// TIA Portal V18 export
FUNCTION_BLOCK "Utility_selection"   // FB7, FBD
TITLE = Selection1_12 , flushing13
{ S7_Optimized_Access := 'TRUE' }
VERSION : 0.1
// stored: AutoNumber false, IsIECCheckEnabled false, IsRetainMemResEnabled false, MemoryReserve 100, SetENOAutomatically false, UDAEnableTagReadback false
   VAR_INPUT
      utl_type : Int;
      chbs_ofb : Bool;
      chbs_cfb : Bool;
      chws_ofb : Bool;
      chws_cfb : Bool;
      cws_ofb : Bool;
      cws_cfb : Bool;
      hws_ofb : Bool;
      hws_cfb : Bool;
      as_ofb : Bool;
      as_cfb : Bool;
      byp_ofb : Bool;
      byp_cfb : Bool;
      chbr_ofb : Bool;
      chbr_cfb : Bool;
      chwr_ofb : Bool;
      chwr_cfb : Bool;
      hwr_ofb : Bool;
      hwr_cfb : Bool;
      cwr_ofb : Bool;
      cwr_cfb : Bool;
      cond_ofb : Bool;
      cond_cfb : Bool;
      dr_ofb : Bool;
      dr_cfb : Bool;
      av_ofb : Bool;
      av_cfb : Bool;
      scv_ofb : Bool;
      times : Array[0..2] of DInt;
   END_VAR
   VAR_OUTPUT
      chbs_cmd : Bool;
      chws_cmd : Bool;
      cws_cmd : Bool;
      hws_cmd : Bool;
      as_cmd : Bool;
      byp_cmd : Bool;
      chbr_cmd : Bool;
      chwr_cmd : Bool;
      cwr_cmd : Bool;
      hwr_cmd : Bool;
      cond_cmd : Bool;
      dr_cmd : Bool;
      av_cmd : Bool;
      scv_cmd : Bool;
      flush_time : DInt;
      vent_time : DInt;
      drine_time : DInt;
      CMNR_cmd : Bool;
   END_VAR
   VAR_IN_OUT
      control { ExternalVisible := 'False'} : Word;
      utl_bit : Bool;
   END_VAR
   VAR
      selection : Int;
      br_sel : Bool;
      chw_sel : Bool;
      cw_sel : Bool;
      hw_sel : Bool;
      flush_sel : Bool;
      st_sel : Bool;
      prev_util : Int;
      vent_start : Bool;
      start_temp : Bool;
      start : Bool;
      flush_tm_comp : Bool;
      am : Bool;
      pause : Bool;
      chbr_cmd1 : Bool;
      chbr_cmd2 : Bool;
      agr_fail : Bool;
      hold : Bool;
      hold_t : Bool;
      status : Word;
      steam_flush : Bool;
      SUV_flush : Bool;
      Pres_low : Bool;
      uti_cv : Bool;
      hw_autoflush : Bool;
      emstop : Bool;
      temp : Bool;
      en_flush : Bool;
      dr_start : Bool;
      hwr_cmd1 : Bool;
      hwr_cmd2 : Bool;
      chwr_cmd1 : Bool;
      chwr_cmd2 : Bool;
      cond_cmd1 : Bool;
      cwr_cmd1 : Bool;
      cwr_cmd2 : Bool;
      br_flush : Bool;
      chw_flush : Bool;
      cw_flush : Bool;
      hw_flush : Bool;
      st_flush : Bool;
      byp_cmd2 : Bool;
      Flush_Dint : DInt;
      Flush_Ptime : Time;
      Flush_Etime : Time;
      Flush_TTime : DInt;
      Vent_Etime : Time;
      Vent_TTime : DInt;
      Vent_Ptime : Time;
      Vent_Dint : DInt;
      Cond_Dint : DInt;
      Cond_Ptime : Time;
      Cond_Etime : Time;
      Cond_TTime : DInt;
      reserved : Bool;
      Vent_tm_comp : Bool;
      Cond_tm_comp : Bool;
      US_TOF3 { S7_SetPoint := 'True'} : TOF_TIME;
      US_TON2 { S7_SetPoint := 'True'} : TON_TIME;
      US_TON3 { S7_SetPoint := 'True'} : TON_TIME;
      US_TON4 { S7_SetPoint := 'True'} : TON_TIME;
      US_TON5 { S7_SetPoint := 'True'} : TON_TIME;
      US_TP2 { S7_SetPoint := 'True'} : TP_TIME;
      US_TP3 { S7_SetPoint := 'True'} : TP_TIME;
      US_TP4 { S7_SetPoint := 'True'} : TP_TIME;
      US_TOF1 { S7_SetPoint := 'True'} : TOF_TIME;
      UP_TP6 { S7_SetPoint := 'True'} : TP_TIME;
      US_TP8 { S7_SetPoint := 'True'} : TP_TIME;
      US_TP7 { S7_SetPoint := 'True'} : TP_TIME;
      US_TP9 { S7_SetPoint := 'True'} : TP_TIME;
      UP_TP1 { S7_SetPoint := 'True'} : TP_TIME;
      US_TP10 { S7_SetPoint := 'True'} : TP_TIME;
      US_TOF2 { S7_SetPoint := 'True'} : TOF_TIME;
      US_TOF4 { S7_SetPoint := 'True'} : TOF_TIME;
      US_TOF6 { S7_SetPoint := 'True'} : TOF_TIME;
      US_TP11 { S7_SetPoint := 'True'} : TP_TIME;
      US_TP12 { S7_SetPoint := 'True'} : TP_TIME;
      US_TON6 { S7_SetPoint := 'True'} : TON_TIME;
      US_TP5 { S7_SetPoint := 'True'} : TP_TIME;
      US_TON7 { S7_SetPoint := 'True'} : TON_TIME;
      US_TP13 { S7_SetPoint := 'True'} : TP_TIME;
      US_TP14 { S7_SetPoint := 'True'} : TP_TIME;
      US_TON8 { S7_SetPoint := 'True'} : TON_TIME;
      US_TP15 { S7_SetPoint := 'True'} : TP_TIME;
      US_TP20 { S7_SetPoint := 'True'} : TP_TIME;
      US_TON10 { S7_SetPoint := 'True'} : TON_TIME;
      US_TP16 { S7_SetPoint := 'True'} : TP_TIME;
      US_TON9 { S7_SetPoint := 'True'} : TON_TIME;
      US_TP17 { S7_SetPoint := 'True'} : TP_TIME;
      US_TP21 { S7_SetPoint := 'True'} : TP_TIME;
      S_TON11 { S7_SetPoint := 'True'} : TON_TIME;
      US_TP18 { S7_SetPoint := 'True'} : TP_TIME;
      US_TP19 { S7_SetPoint := 'True'} : TP_TIME;
   END_VAR
   VAR_TEMP   // added for the SCL form of the ladder/FBD networks
      _w1 : Bool;
   END_VAR
BEGIN

REGION Network 1: utility selection and moving
   // utility selection and moving
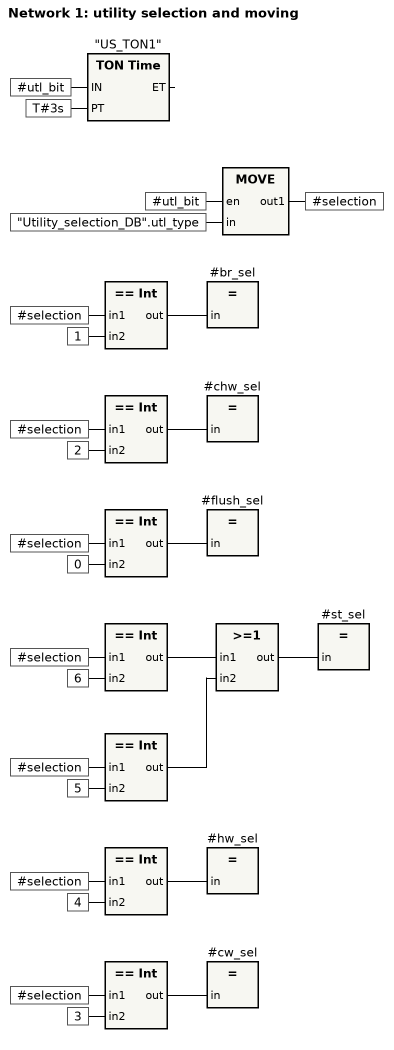
   "US_TON1".TON(IN := #utl_bit, PT := T#3s);
   IF #utl_bit THEN #selection := "Utility_selection_DB".utl_type; END_IF;
   #br_sel := #selection = 1;
   #chw_sel := #selection = 2;
   #flush_sel := #selection = 0;
   #st_sel := (#selection = 6) OR (#selection = 5);
   #hw_sel := #selection = 4;
   #cw_sel := #selection = 3;
END_REGION

REGION Network 2: previous utiliy identifucation
   // previous utiliy identifucation
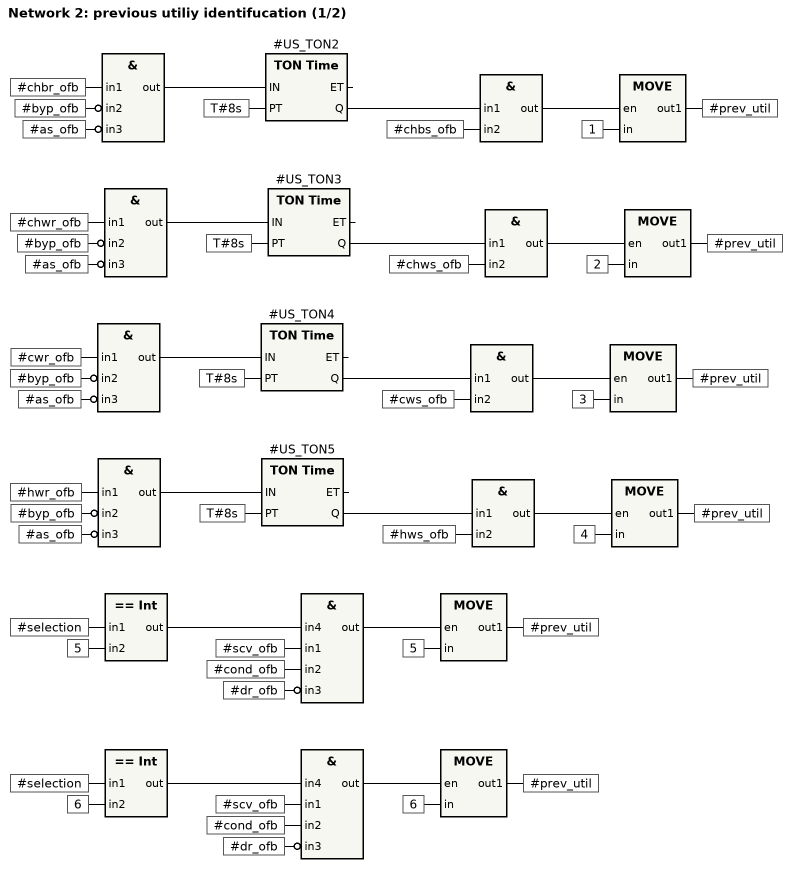
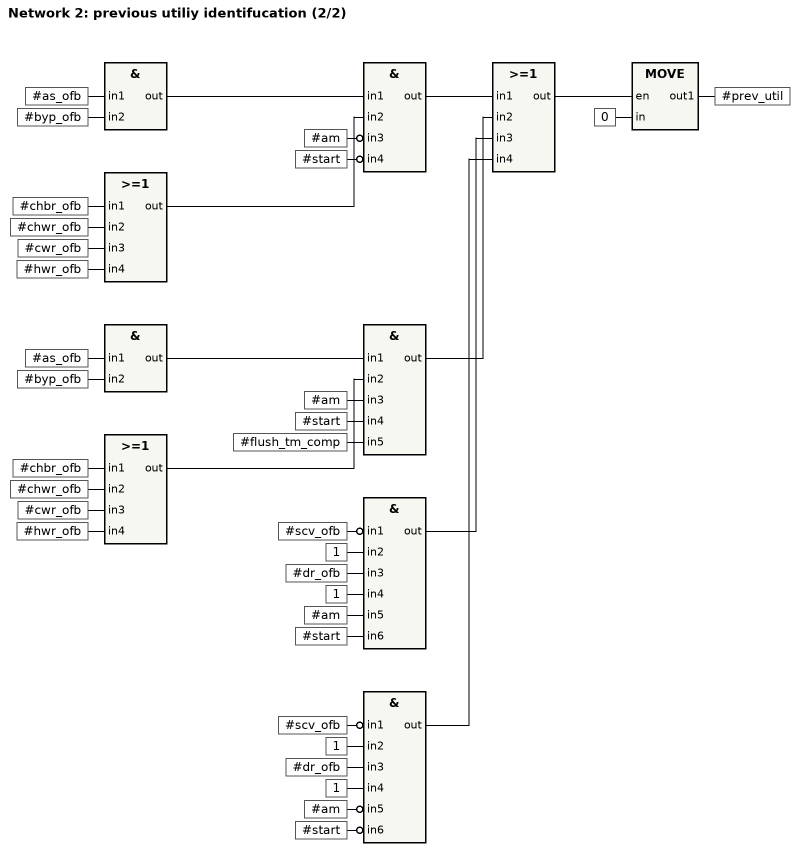
   #US_TON2(IN := #chbr_ofb AND NOT #byp_ofb AND NOT #as_ofb, PT := T#8s);   // TON
   IF #US_TON2.Q AND #chbs_ofb THEN #prev_util := 1; END_IF;
   #US_TON3(IN := #chwr_ofb AND NOT #byp_ofb AND NOT #as_ofb, PT := T#8s);   // TON
   IF #US_TON3.Q AND #chws_ofb THEN #prev_util := 2; END_IF;
   #US_TON4(IN := #cwr_ofb AND NOT #byp_ofb AND NOT #as_ofb, PT := T#8s);   // TON
   IF #US_TON4.Q AND #cws_ofb THEN #prev_util := 3; END_IF;
   #US_TON5(IN := #hwr_ofb AND NOT #byp_ofb AND NOT #as_ofb, PT := T#8s);   // TON
   IF #US_TON5.Q AND #hws_ofb THEN #prev_util := 4; END_IF;
   IF (#selection = 5) AND #scv_ofb AND #cond_ofb AND NOT #dr_ofb THEN #prev_util := 5; END_IF;
   IF (#selection = 6) AND #scv_ofb AND #cond_ofb AND NOT #dr_ofb THEN #prev_util := 6; END_IF;
   IF (#as_ofb AND #byp_ofb AND (#chbr_ofb OR #chwr_ofb OR #cwr_ofb OR #hwr_ofb) AND NOT #am AND NOT #start) OR (#as_ofb AND #byp_ofb AND (#chbr_ofb OR #chwr_ofb OR #cwr_ofb OR #hwr_ofb) AND #am AND #start AND #flush_tm_comp) OR (NOT #scv_ofb AND 1 AND #dr_ofb AND 1 AND #am AND #start) OR (NOT #scv_ofb AND 1 AND #dr_ofb AND 1 AND NOT #am AND NOT #start) THEN
       #prev_util := 0;
   END_IF;
END_REGION

REGION Network 3: flushing Identification
   // flushing Identification
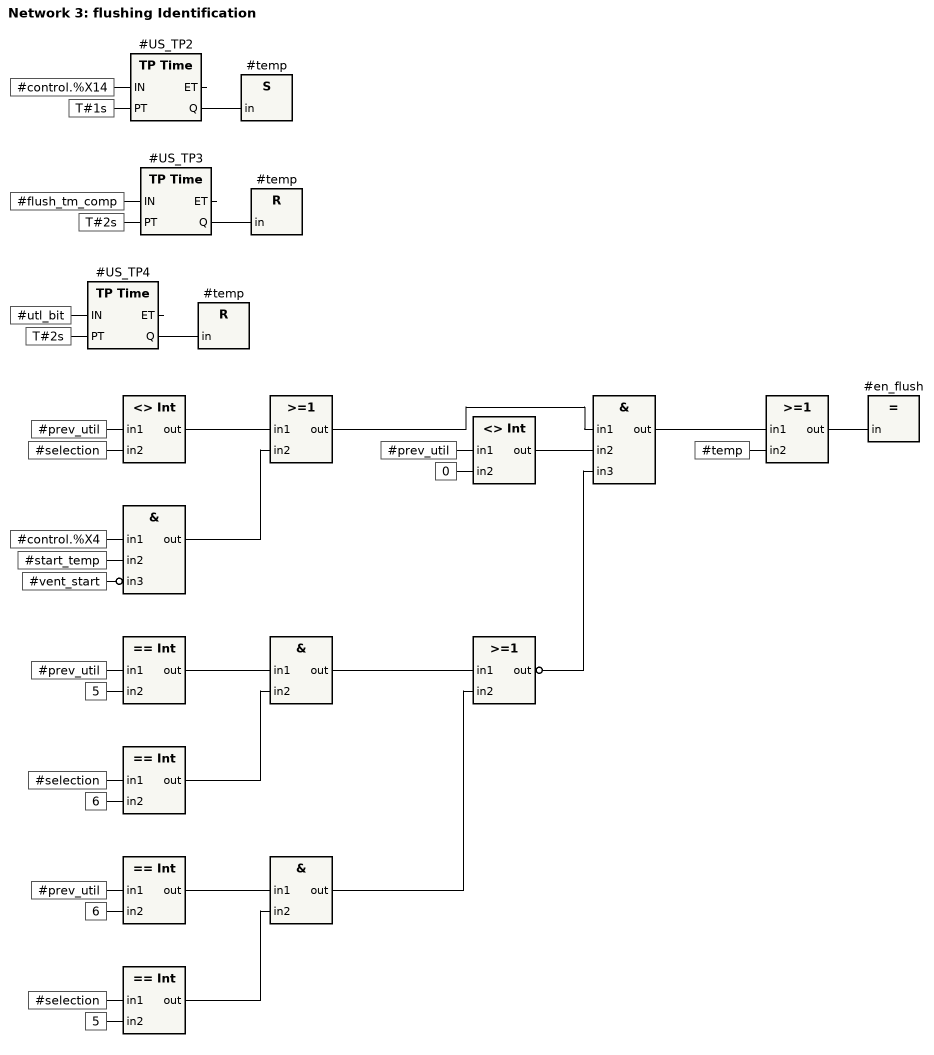
   #US_TP2(IN := #control.%X14, PT := T#1s);   // TP
   IF #US_TP2.Q THEN #temp := TRUE; END_IF;
   #US_TP3(IN := #flush_tm_comp, PT := T#2s);   // TP
   IF #US_TP3.Q THEN #temp := FALSE; END_IF;
   #US_TP4(IN := #utl_bit, PT := T#2s);   // TP
   IF #US_TP4.Q THEN #temp := FALSE; END_IF;
   #en_flush := (((#prev_util <> #selection) OR (#control.%X4 AND #start_temp AND NOT #vent_start)) AND (#prev_util <> 0) AND NOT (((#prev_util = 5) AND (#selection = 6)) OR ((#prev_util = 6) AND (#selection = 5)))) OR #temp;
END_REGION

REGION Network 4: temp_start
   // temp_start
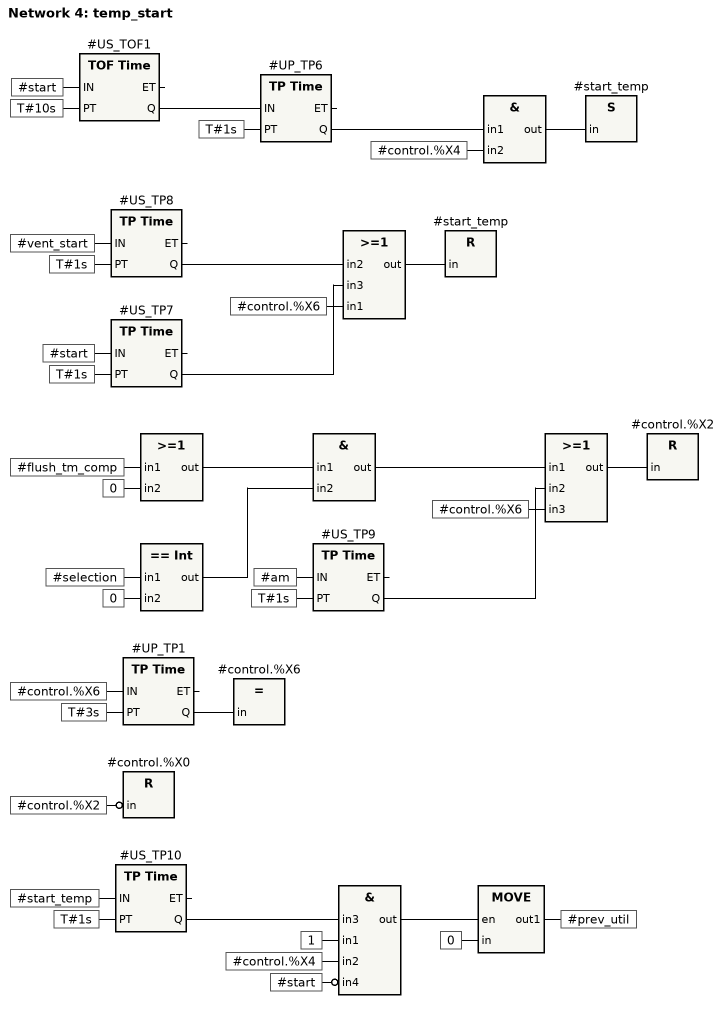
   #US_TOF1(IN := #start, PT := T#10s);   // TOF
   #UP_TP6(IN := #US_TOF1.Q, PT := T#1s);   // TP
   IF #UP_TP6.Q AND #control.%X4 THEN #start_temp := TRUE; END_IF;
   #US_TP8(IN := #vent_start, PT := T#1s);   // TP
   #US_TP7(IN := #start, PT := T#1s);   // TP
   IF #US_TP8.Q OR #US_TP7.Q OR #control.%X6 THEN #start_temp := FALSE; END_IF;
   #US_TP9(IN := #am, PT := T#1s);   // TP
   IF ((#flush_tm_comp OR 0) AND (#selection = 0)) OR #US_TP9.Q OR #control.%X6 THEN
       #control.%X2 := FALSE;
   END_IF;
   #UP_TP1(IN := #control.%X6, PT := T#3s);   // TP
   #control.%X6 := #UP_TP1.Q;
   IF NOT #control.%X2 THEN #control.%X0 := FALSE; END_IF;
   #US_TP10(IN := #start_temp, PT := T#1s);   // TP
   IF #US_TP10.Q AND 1 AND #control.%X4 AND NOT #start THEN #prev_util := 0; END_IF;
END_REGION

REGION Network 5: control and status word
   // control and status word
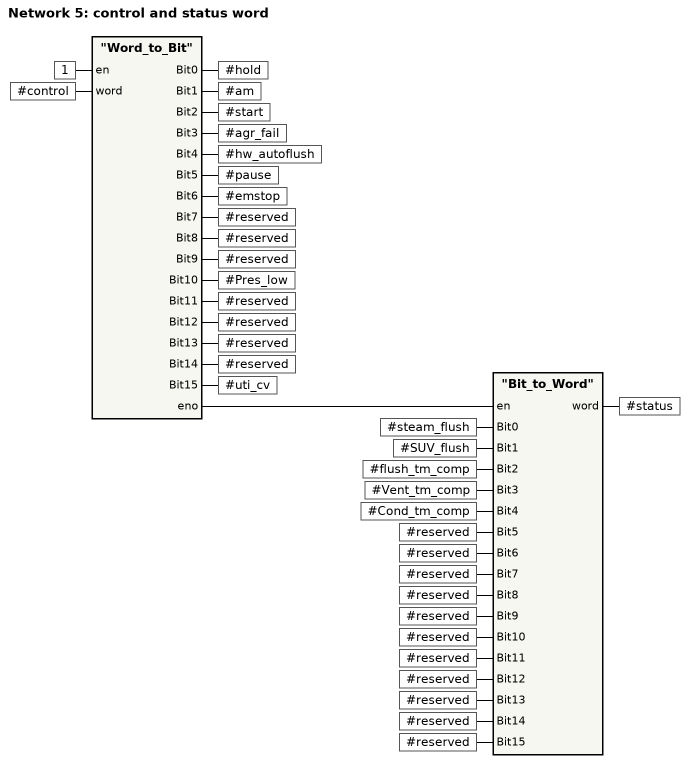
   "Word_to_Bit"(EN := 1,
                 "word" := #control,
                 Bit0 => #hold,
                 Bit1 => #am,
                 Bit2 => #start,
                 Bit3 => #agr_fail,
                 Bit4 => #hw_autoflush,
                 Bit5 => #pause,
                 Bit6 => #emstop,
                 Bit7 => #reserved,
                 Bit8 => #reserved,
                 Bit9 => #reserved,
                 Bit10 => #Pres_low,
                 Bit11 => #reserved,
                 Bit12 => #reserved,
                 Bit13 => #reserved,
                 Bit14 => #reserved,
                 Bit15 => #uti_cv,
                 ENO => #_w1);
   IF #_w1 THEN
       "Bit_to_Word"(Bit0 := #steam_flush,
                     Bit1 := #SUV_flush,
                     Bit2 := #flush_tm_comp,
                     Bit3 := #Vent_tm_comp,
                     Bit4 := #Cond_tm_comp,
                     Bit5 := #reserved,
                     Bit6 := #reserved,
                     Bit7 := #reserved,
                     Bit8 := #reserved,
                     Bit9 := #reserved,
                     Bit10 := #reserved,
                     Bit11 := #reserved,
                     Bit12 := #reserved,
                     Bit13 := #reserved,
                     Bit14 := #reserved,
                     Bit15 := #reserved,
                     "word" => #status);
   END_IF;
END_REGION

REGION Network 6: Brine select
   // Brine select
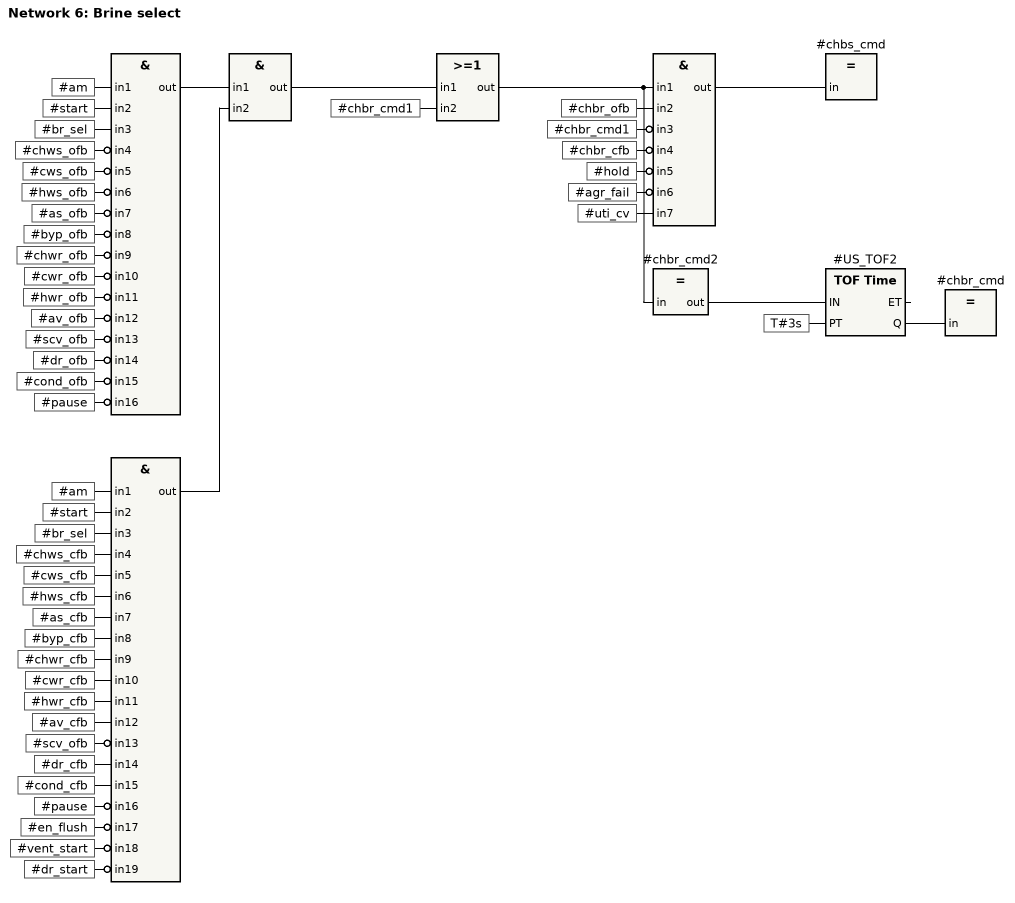
   #_w1 := (#am AND #start AND #br_sel AND NOT #chws_ofb AND NOT #cws_ofb AND NOT #hws_ofb AND NOT #as_ofb AND NOT #byp_ofb AND NOT #chwr_ofb AND NOT #cwr_ofb AND NOT #hwr_ofb AND NOT #av_ofb AND NOT #scv_ofb AND NOT #dr_ofb AND NOT #cond_ofb AND NOT #pause AND #am AND #start AND #br_sel AND #chws_cfb AND #cws_cfb AND #hws_cfb AND #as_cfb AND #byp_cfb AND #chwr_cfb AND #cwr_cfb AND #hwr_cfb AND #av_cfb AND NOT #scv_ofb AND #dr_cfb AND #cond_cfb AND NOT #pause AND NOT #en_flush AND NOT #vent_start AND NOT #dr_start) OR #chbr_cmd1;
   #chbs_cmd := #_w1 AND #chbr_ofb AND NOT #chbr_cmd1 AND NOT #chbr_cfb AND NOT #hold AND NOT #agr_fail AND #uti_cv;
   #chbr_cmd2 := #_w1;
   #US_TOF2(IN := #_w1, PT := T#3s);   // TOF
   #chbr_cmd := #US_TOF2.Q;
END_REGION

REGION Network 7: CMNR logic
   // CMNR logic
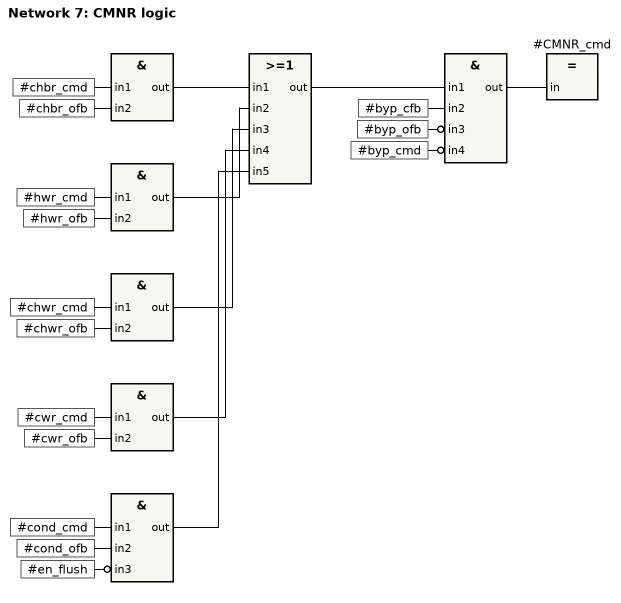
   #CMNR_cmd := ((#chbr_cmd AND #chbr_ofb) OR (#hwr_cmd AND #hwr_ofb) OR (#chwr_cmd AND #chwr_ofb) OR (#cwr_cmd AND #cwr_ofb) OR (#cond_cmd AND #cond_ofb AND NOT #en_flush)) AND #byp_cfb AND NOT #byp_ofb AND NOT #byp_cmd;
END_REGION

REGION Network 8: HW select
   // Hw select
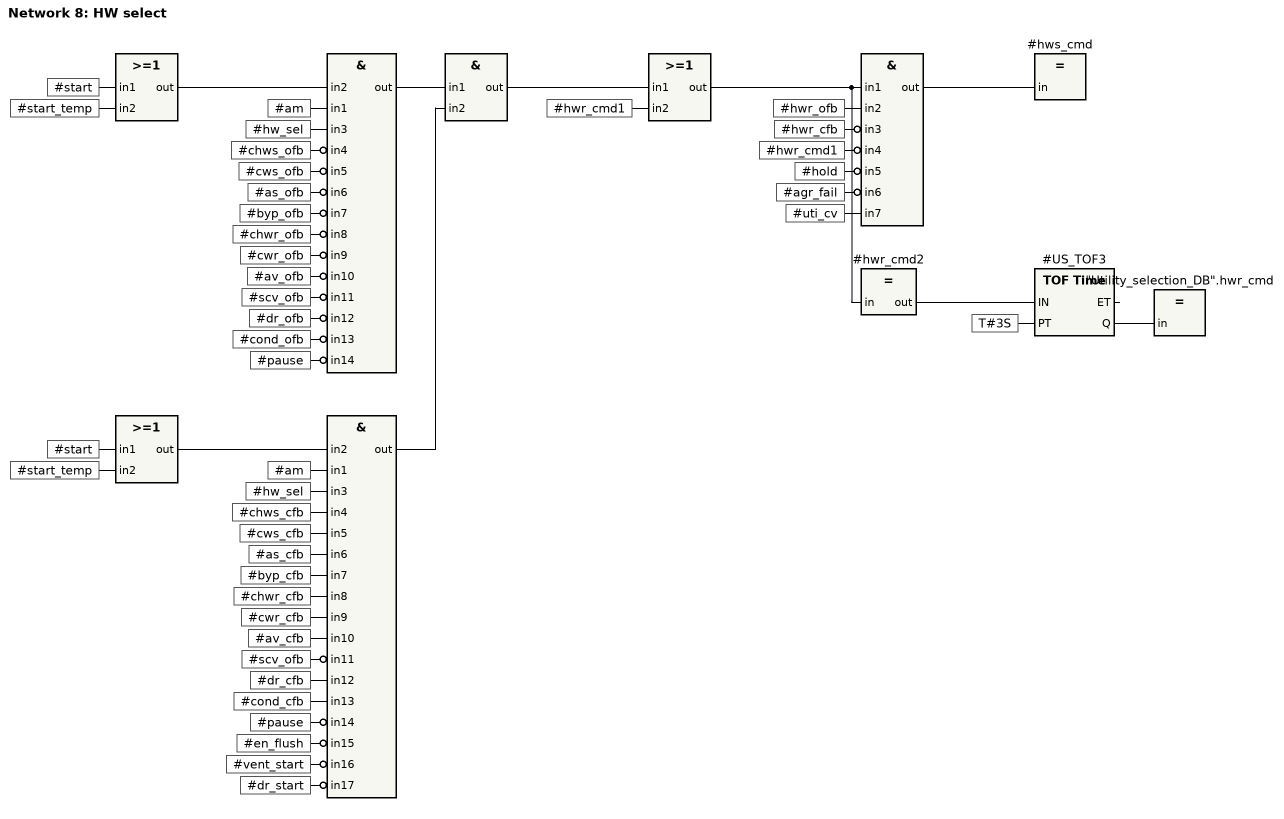
   #_w1 := ((#start OR #start_temp) AND #am AND #hw_sel AND NOT #chws_ofb AND NOT #cws_ofb AND NOT #as_ofb AND NOT #byp_ofb AND NOT #chwr_ofb AND NOT #cwr_ofb AND NOT #av_ofb AND NOT #scv_ofb AND NOT #dr_ofb AND NOT #cond_ofb AND NOT #pause AND (#start OR #start_temp) AND #am AND #hw_sel AND #chws_cfb AND #cws_cfb AND #as_cfb AND #byp_cfb AND #chwr_cfb AND #cwr_cfb AND #av_cfb AND NOT #scv_ofb AND #dr_cfb AND #cond_cfb AND NOT #pause AND NOT #en_flush AND NOT #vent_start AND NOT #dr_start) OR #hwr_cmd1;
   #hws_cmd := #_w1 AND #hwr_ofb AND NOT #hwr_cfb AND NOT #hwr_cmd1 AND NOT #hold AND NOT #agr_fail AND #uti_cv;
   #hwr_cmd2 := #_w1;
   #US_TOF3(IN := #_w1, PT := T#3S);   // TOF
   "Utility_selection_DB".hwr_cmd := #US_TOF3.Q;
END_REGION

REGION Network 9: chw select
   // chw select
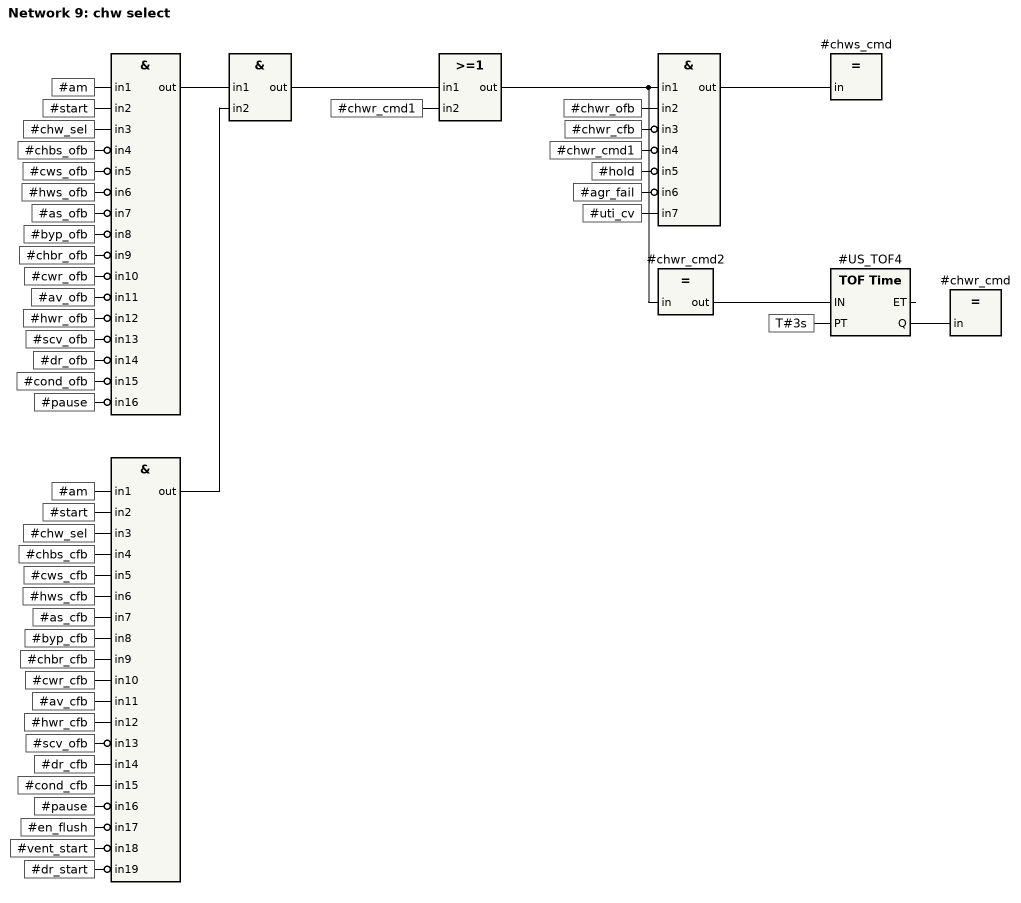
   #_w1 := (#am AND #start AND #chw_sel AND NOT #chbs_ofb AND NOT #cws_ofb AND NOT #hws_ofb AND NOT #as_ofb AND NOT #byp_ofb AND NOT #chbr_ofb AND NOT #cwr_ofb AND NOT #av_ofb AND NOT #hwr_ofb AND NOT #scv_ofb AND NOT #dr_ofb AND NOT #cond_ofb AND NOT #pause AND #am AND #start AND #chw_sel AND #chbs_cfb AND #cws_cfb AND #hws_cfb AND #as_cfb AND #byp_cfb AND #chbr_cfb AND #cwr_cfb AND #av_cfb AND #hwr_cfb AND NOT #scv_ofb AND #dr_cfb AND #cond_cfb AND NOT #pause AND NOT #en_flush AND NOT #vent_start AND NOT #dr_start) OR #chwr_cmd1;
   #chws_cmd := #_w1 AND #chwr_ofb AND NOT #chwr_cfb AND NOT #chwr_cmd1 AND NOT #hold AND NOT #agr_fail AND #uti_cv;
   #chwr_cmd2 := #_w1;
   #US_TOF4(IN := #_w1, PT := T#3s);   // TOF
   #chwr_cmd := #US_TOF4.Q;
END_REGION

REGION Network 10: Steam select
   // Steam select
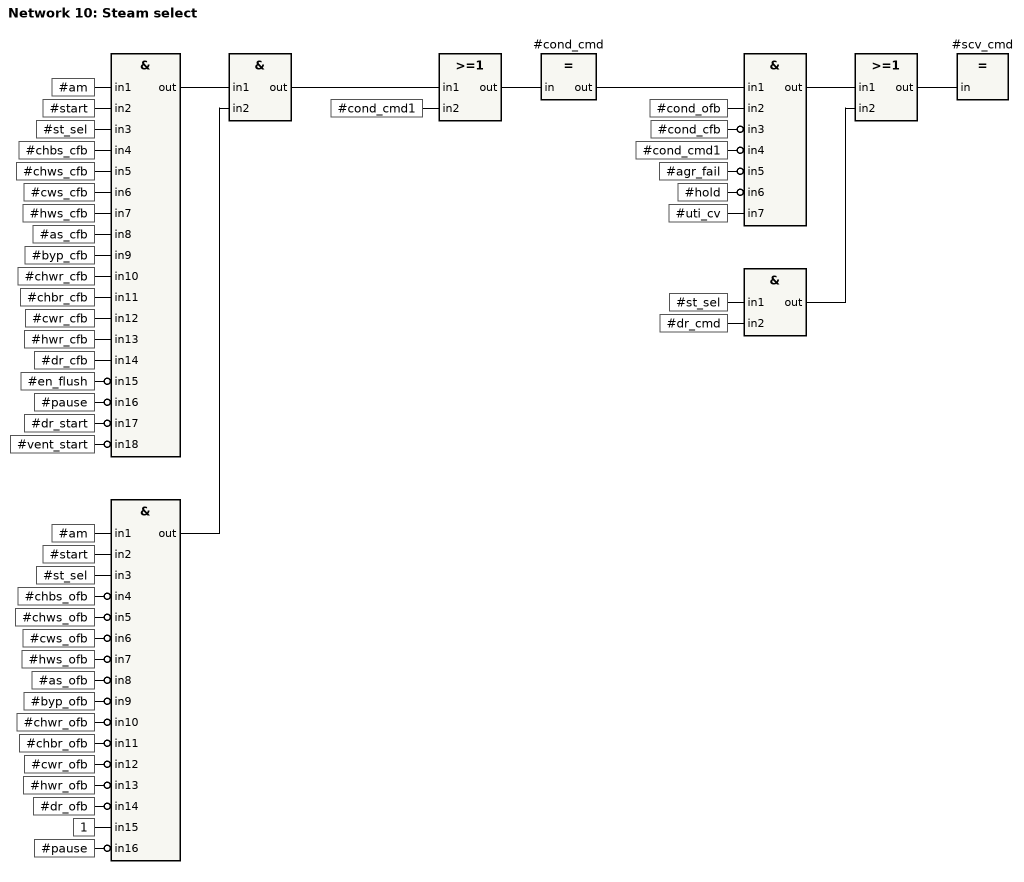
   #cond_cmd := (#am AND #start AND #st_sel AND #chbs_cfb AND #chws_cfb AND #cws_cfb AND #hws_cfb AND #as_cfb AND #byp_cfb AND #chwr_cfb AND #chbr_cfb AND #cwr_cfb AND #hwr_cfb AND #dr_cfb AND NOT #en_flush AND NOT #pause AND NOT #dr_start AND NOT #vent_start AND #am AND #start AND #st_sel AND NOT #chbs_ofb AND NOT #chws_ofb AND NOT #cws_ofb AND NOT #hws_ofb AND NOT #as_ofb AND NOT #byp_ofb AND NOT #chwr_ofb AND NOT #chbr_ofb AND NOT #cwr_ofb AND NOT #hwr_ofb AND NOT #dr_ofb AND 1 AND NOT #pause) OR #cond_cmd1;
   #scv_cmd := (#cond_cmd AND #cond_ofb AND NOT #cond_cfb AND NOT #cond_cmd1 AND NOT #agr_fail AND NOT #hold AND #uti_cv) OR (#st_sel AND #dr_cmd);
END_REGION

REGION Network 11: cw_select
   // cw_select
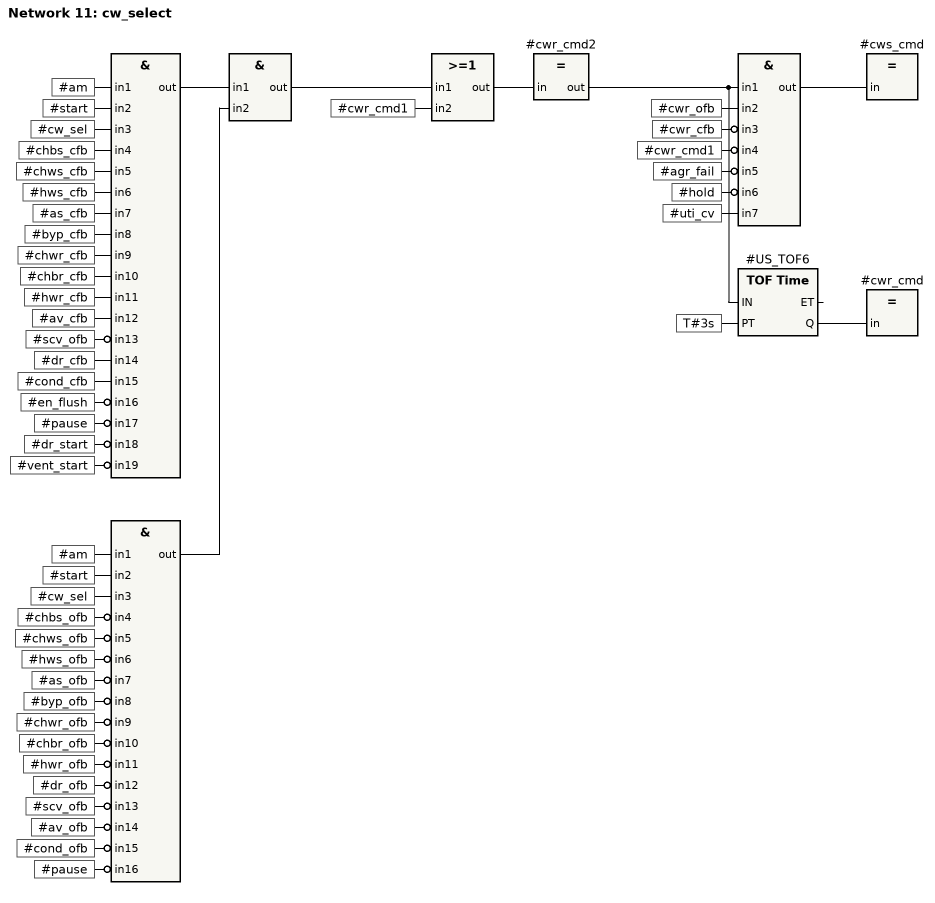
   #cwr_cmd2 := (#am AND #start AND #cw_sel AND #chbs_cfb AND #chws_cfb AND #hws_cfb AND #as_cfb AND #byp_cfb AND #chwr_cfb AND #chbr_cfb AND #hwr_cfb AND #av_cfb AND NOT #scv_ofb AND #dr_cfb AND #cond_cfb AND NOT #en_flush AND NOT #pause AND NOT #dr_start AND NOT #vent_start AND #am AND #start AND #cw_sel AND NOT #chbs_ofb AND NOT #chws_ofb AND NOT #hws_ofb AND NOT #as_ofb AND NOT #byp_ofb AND NOT #chwr_ofb AND NOT #chbr_ofb AND NOT #hwr_ofb AND NOT #dr_ofb AND NOT #scv_ofb AND NOT #av_ofb AND NOT #cond_ofb AND NOT #pause) OR #cwr_cmd1;
   #cws_cmd := #cwr_cmd2 AND #cwr_ofb AND NOT #cwr_cfb AND NOT #cwr_cmd1 AND NOT #agr_fail AND NOT #hold AND #uti_cv;
   #US_TOF6(IN := #cwr_cmd2, PT := T#3s);   // TOF
   #cwr_cmd := #US_TOF6.Q;
END_REGION

REGION Network 12: flush selection
   // flush selection
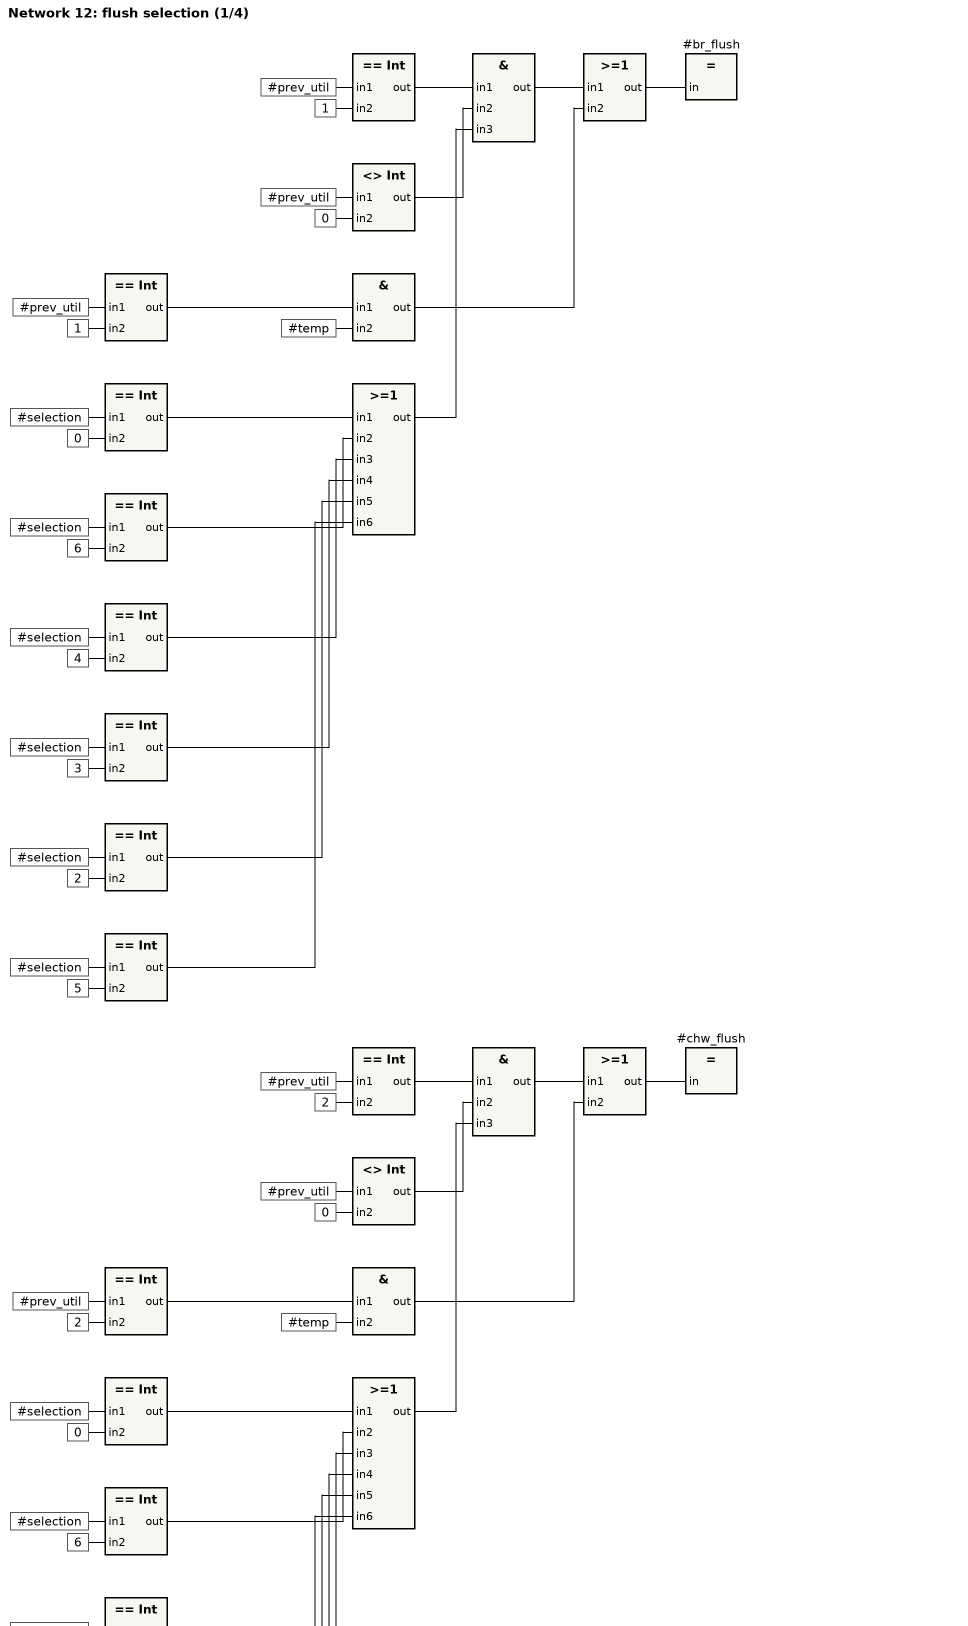
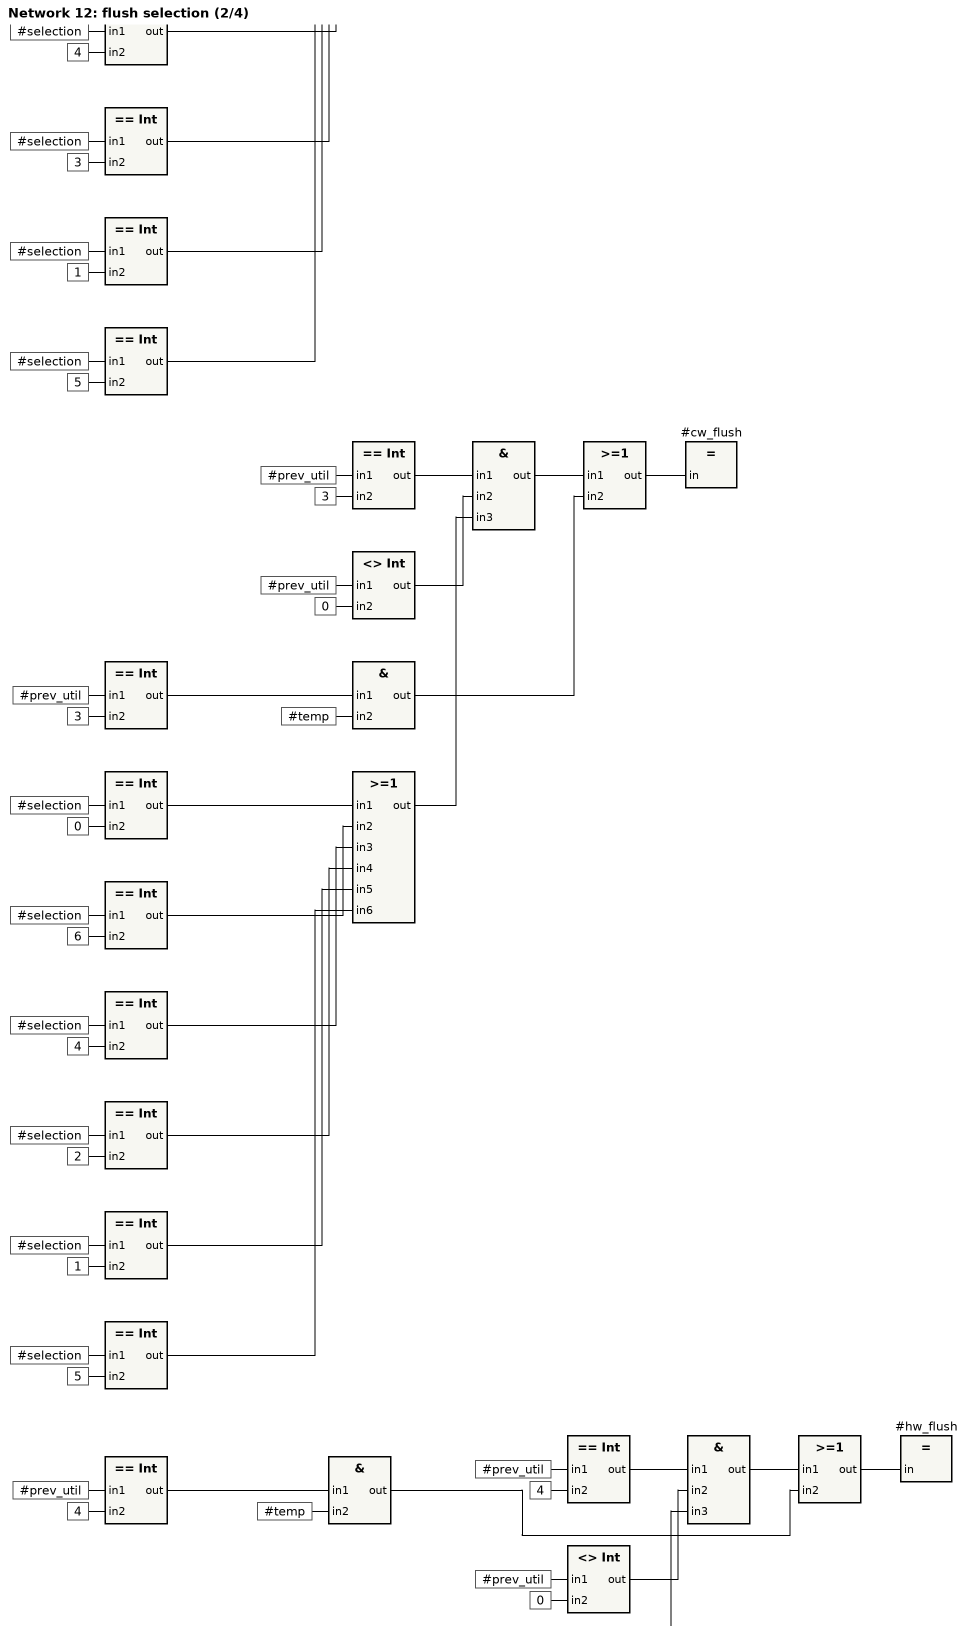
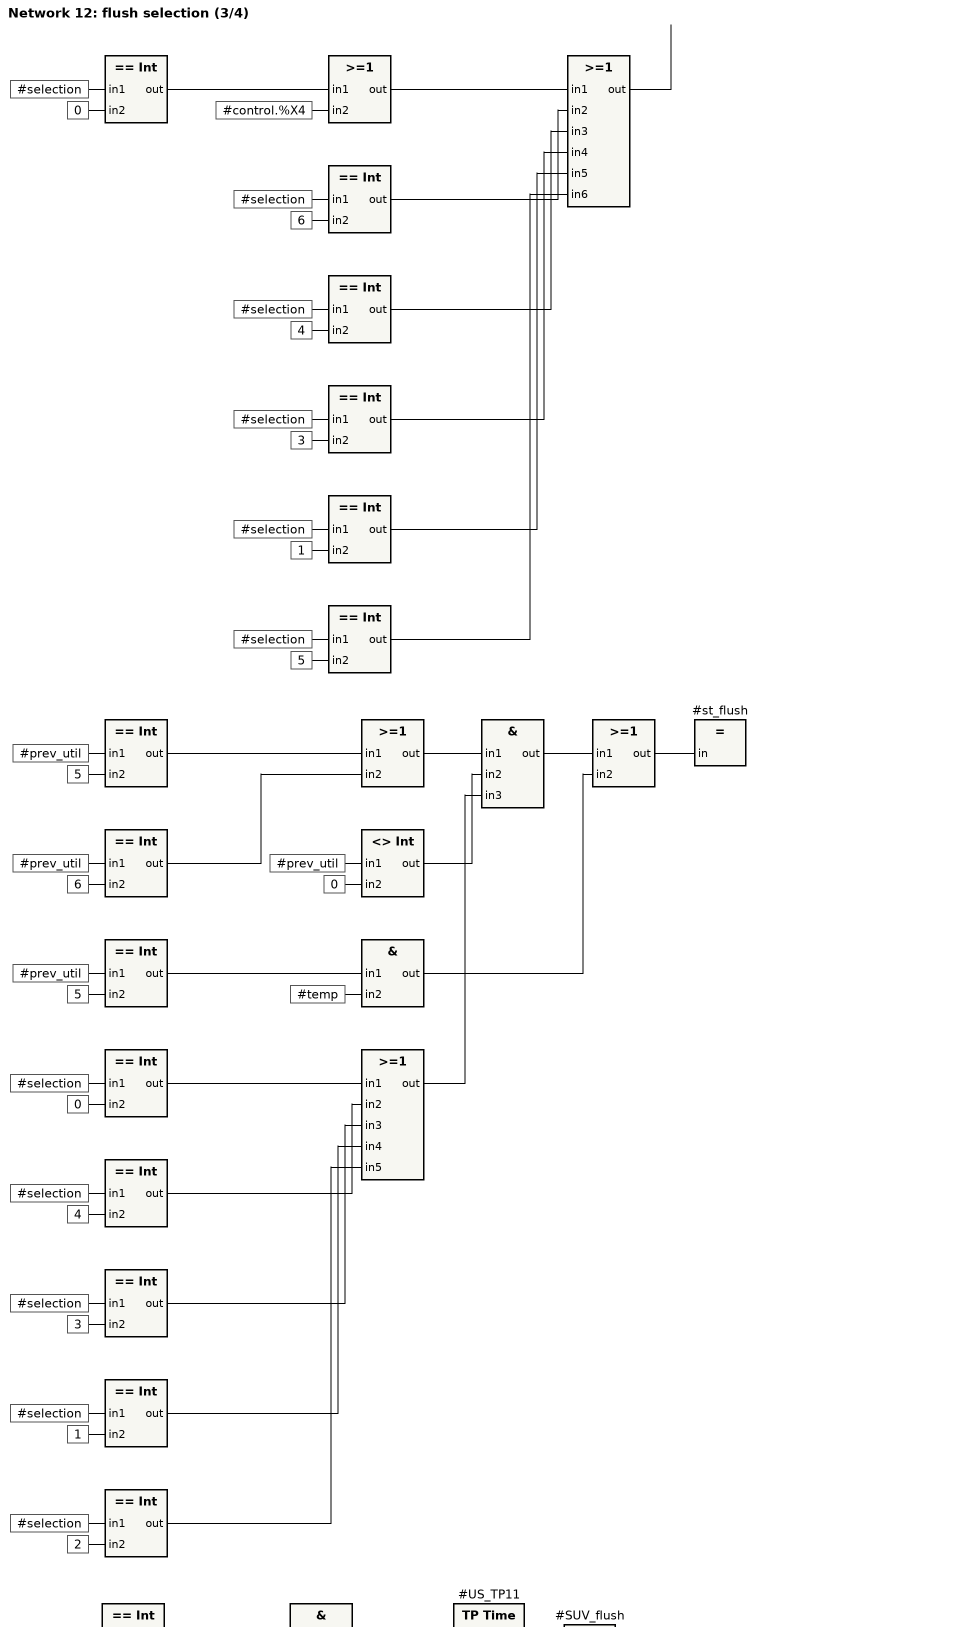
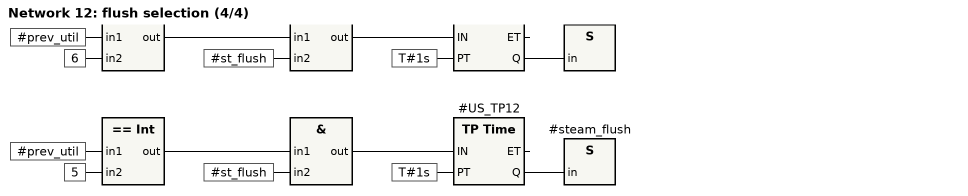
   #br_flush := ((#prev_util = 1) AND (#prev_util <> 0) AND ((#selection = 0) OR (#selection = 6) OR (#selection = 4) OR (#selection = 3) OR (#selection = 2) OR (#selection = 5))) OR ((#prev_util = 1) AND #temp);
   #chw_flush := ((#prev_util = 2) AND (#prev_util <> 0) AND ((#selection = 0) OR (#selection = 6) OR (#selection = 4) OR (#selection = 3) OR (#selection = 1) OR (#selection = 5))) OR ((#prev_util = 2) AND #temp);
   #cw_flush := ((#prev_util = 3) AND (#prev_util <> 0) AND ((#selection = 0) OR (#selection = 6) OR (#selection = 4) OR (#selection = 2) OR (#selection = 1) OR (#selection = 5))) OR ((#prev_util = 3) AND #temp);
   #hw_flush := ((#prev_util = 4) AND (#prev_util <> 0) AND ((#selection = 0) OR #control.%X4 OR (#selection = 6) OR (#selection = 4) OR (#selection = 3) OR (#selection = 1) OR (#selection = 5))) OR ((#prev_util = 4) AND #temp);
   #st_flush := (((#prev_util = 5) OR (#prev_util = 6)) AND (#prev_util <> 0) AND ((#selection = 0) OR (#selection = 4) OR (#selection = 3) OR (#selection = 1) OR (#selection = 2))) OR ((#prev_util = 5) AND #temp);
   #US_TP11(IN := (#prev_util = 6) AND #st_flush, PT := T#1s);   // TP
   IF #US_TP11.Q THEN #SUV_flush := TRUE; END_IF;
   #US_TP12(IN := (#prev_util = 5) AND #st_flush, PT := T#1s);   // TP
   IF #US_TP12.Q THEN #steam_flush := TRUE; END_IF;
END_REGION

REGION Network 13: Flushing Timer
   // Flushing timer
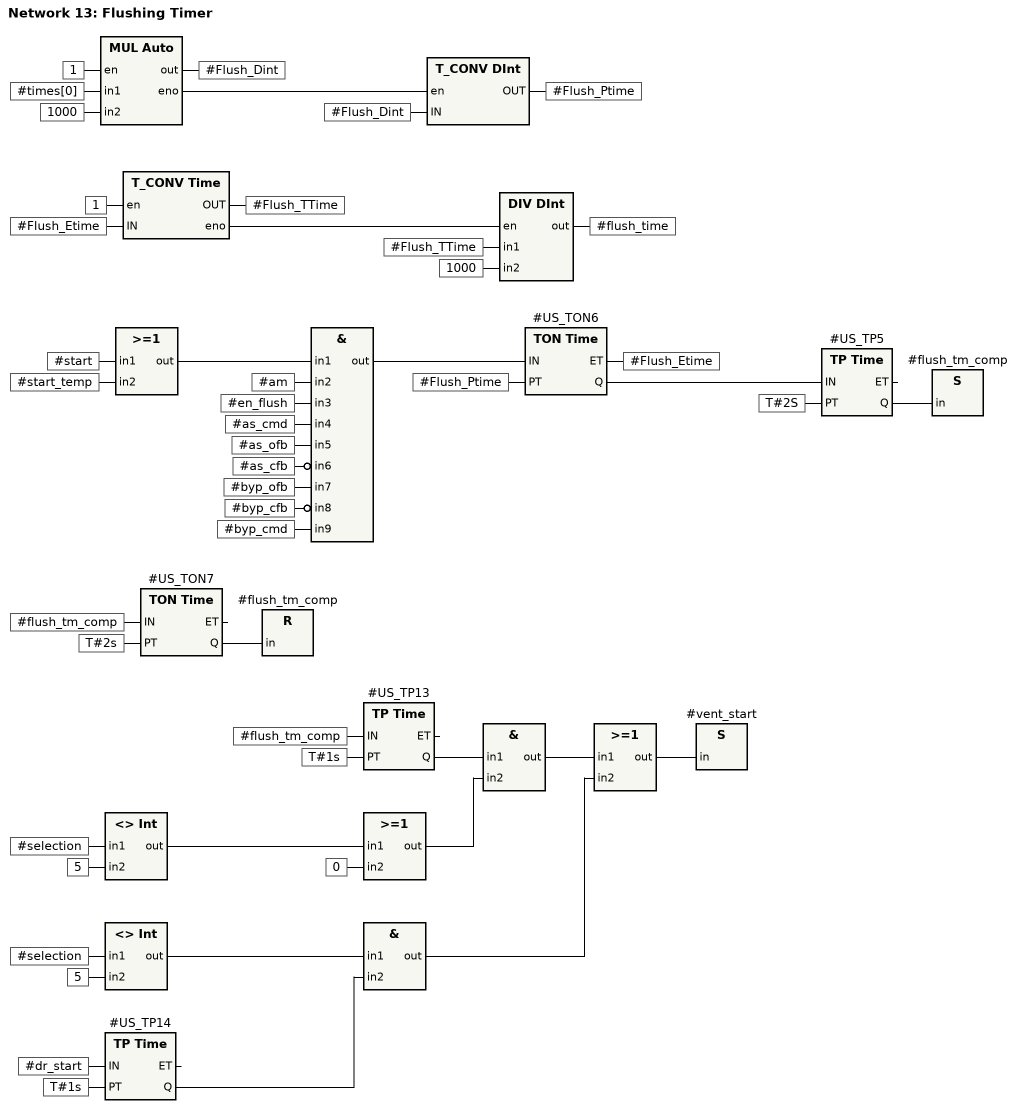
   IF 1 THEN
       #Flush_Dint := #times[0] * 1000;
       T_CONV(IN := #Flush_Dint, OUT => #Flush_Ptime);
   END_IF;
   T_CONV(EN := 1, IN := #Flush_Etime, OUT => #Flush_TTime, ENO => #_w1);
   IF #_w1 THEN #flush_time := #Flush_TTime / 1000; END_IF;
   #US_TON6(IN := (#start OR #start_temp) AND #am AND #en_flush AND #as_cmd AND #as_ofb AND NOT #as_cfb AND #byp_ofb AND NOT #byp_cfb AND #byp_cmd,   // TON
            PT := #Flush_Ptime,
            ET => #Flush_Etime);
   #US_TP5(IN := #US_TON6.Q, PT := T#2S);   // TP
   IF #US_TP5.Q THEN #flush_tm_comp := TRUE; END_IF;
   #US_TON7(IN := #flush_tm_comp, PT := T#2s);   // TON
   IF #US_TON7.Q THEN #flush_tm_comp := FALSE; END_IF;
   #US_TP13(IN := #flush_tm_comp, PT := T#1s);   // TP
   #US_TP14(IN := #dr_start, PT := T#1s);   // TP
   IF (#US_TP13.Q AND ((#selection <> 5) OR 0)) OR ((#selection <> 5) AND #US_TP14.Q) THEN
       #vent_start := TRUE;
   END_IF;
END_REGION

REGION Network 14: vent timer
   // vent timer
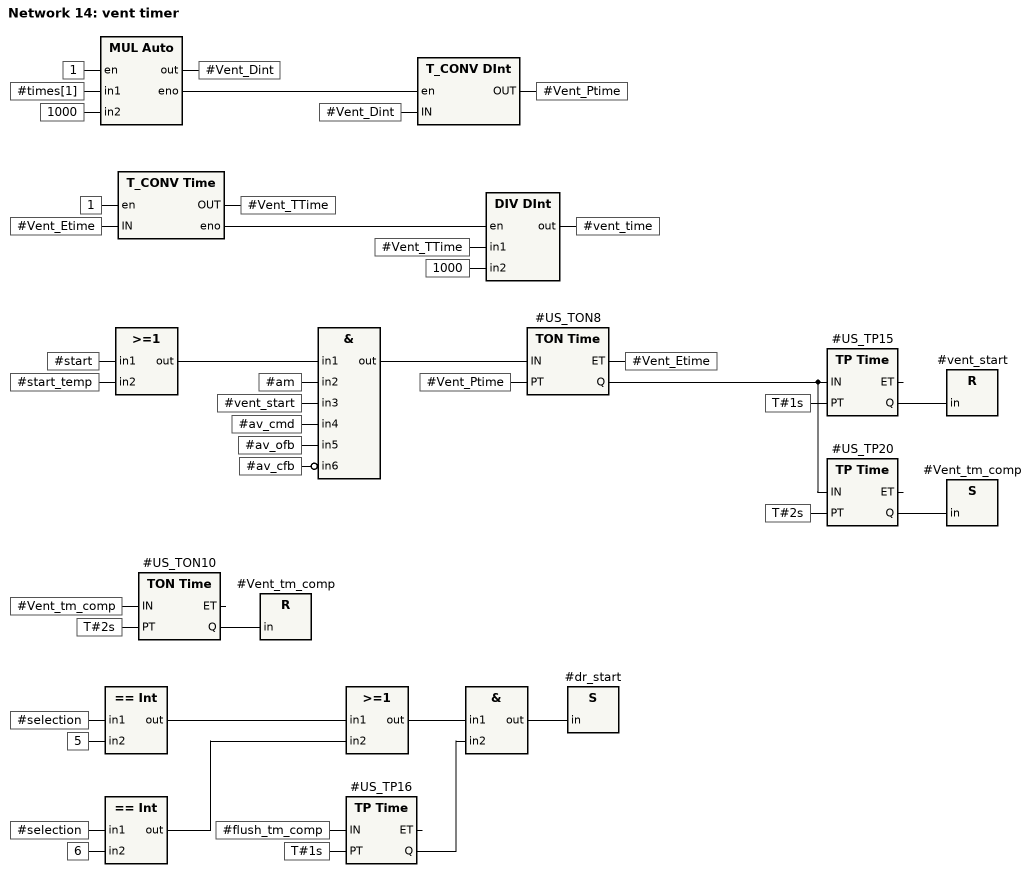
   IF 1 THEN
       #Vent_Dint := #times[1] * 1000;
       T_CONV(IN := #Vent_Dint, OUT => #Vent_Ptime);
   END_IF;
   T_CONV(EN := 1, IN := #Vent_Etime, OUT => #Vent_TTime, ENO => #_w1);
   IF #_w1 THEN #vent_time := #Vent_TTime / 1000; END_IF;
   #US_TON8(IN := (#start OR #start_temp) AND #am AND #vent_start AND #av_cmd AND #av_ofb AND NOT #av_cfb,   // TON
            PT := #Vent_Ptime,
            ET => #Vent_Etime);
   #US_TP15(IN := #US_TON8.Q, PT := T#1s);   // TP
   IF #US_TP15.Q THEN #vent_start := FALSE; END_IF;
   #US_TP20(IN := #US_TON8.Q, PT := T#2s);   // TP
   IF #US_TP20.Q THEN #Vent_tm_comp := TRUE; END_IF;
   #US_TON10(IN := #Vent_tm_comp, PT := T#2s);   // TON
   IF #US_TON10.Q THEN #Vent_tm_comp := FALSE; END_IF;
   #US_TP16(IN := #flush_tm_comp, PT := T#1s);   // TP
   IF ((#selection = 5) OR (#selection = 6)) AND #US_TP16.Q THEN #dr_start := TRUE; END_IF;
END_REGION

REGION Network 15: Condensation timer
   // condensation timer
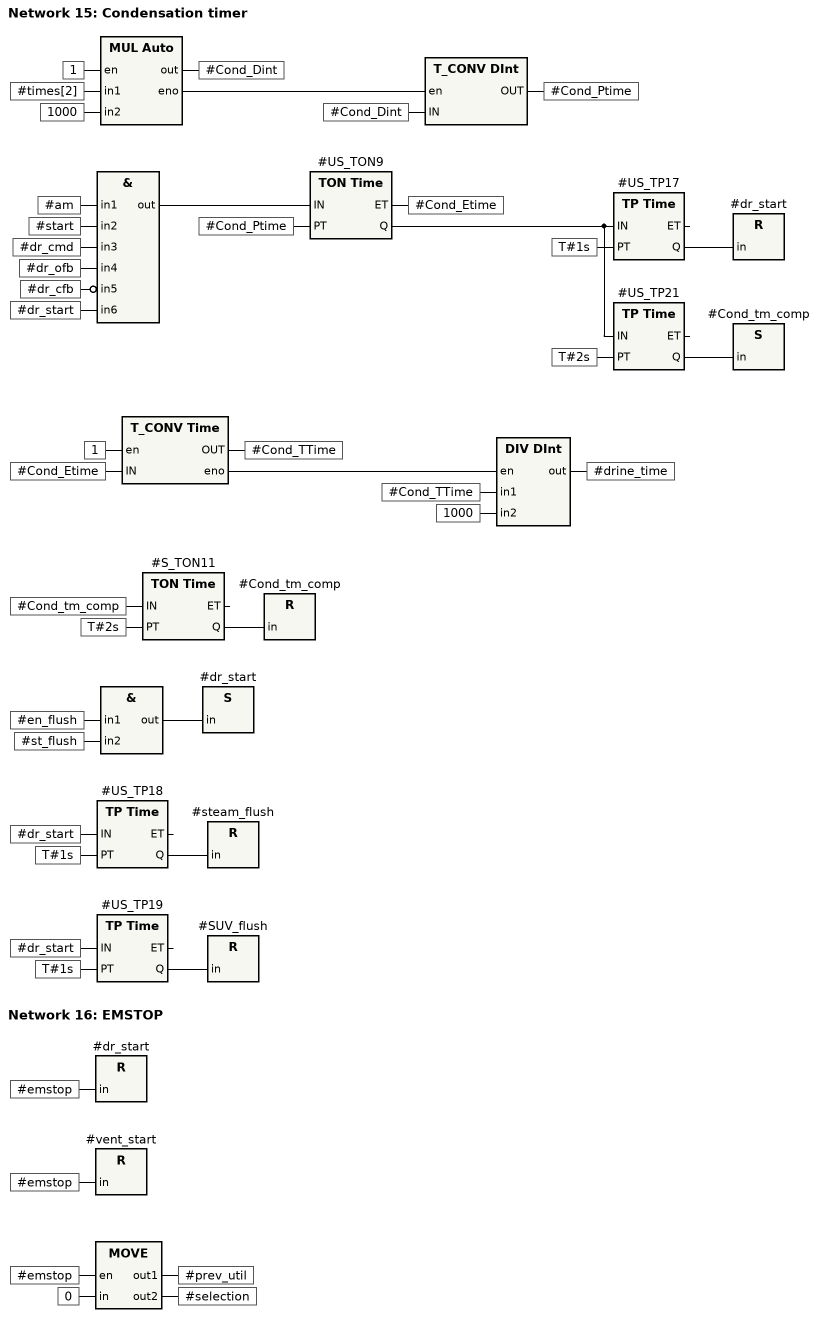
   IF 1 THEN
       #Cond_Dint := #times[2] * 1000;
       T_CONV(IN := #Cond_Dint, OUT => #Cond_Ptime);
   END_IF;
   #US_TON9(IN := #am AND #start AND #dr_cmd AND #dr_ofb AND NOT #dr_cfb AND #dr_start,   // TON
            PT := #Cond_Ptime,
            ET => #Cond_Etime);
   #US_TP17(IN := #US_TON9.Q, PT := T#1s);   // TP
   IF #US_TP17.Q THEN #dr_start := FALSE; END_IF;
   #US_TP21(IN := #US_TON9.Q, PT := T#2s);   // TP
   IF #US_TP21.Q THEN #Cond_tm_comp := TRUE; END_IF;
   T_CONV(EN := 1, IN := #Cond_Etime, OUT => #Cond_TTime, ENO => #_w1);
   IF #_w1 THEN #drine_time := #Cond_TTime / 1000; END_IF;
   #S_TON11(IN := #Cond_tm_comp, PT := T#2s);   // TON
   IF #S_TON11.Q THEN #Cond_tm_comp := FALSE; END_IF;
   IF #en_flush AND #st_flush THEN #dr_start := TRUE; END_IF;
   #US_TP18(IN := #dr_start, PT := T#1s);   // TP
   IF #US_TP18.Q THEN #steam_flush := FALSE; END_IF;
   #US_TP19(IN := #dr_start, PT := T#1s);   // TP
   IF #US_TP19.Q THEN #SUV_flush := FALSE; END_IF;
END_REGION

REGION Network 16: EMSTOP
   // EMSTOP
   IF #emstop THEN
       #dr_start := FALSE;
       #vent_start := FALSE;
       #prev_util := 0;
       #selection := 0;
   END_IF;
END_REGION

REGION Network 17: Brine flushing logic
   // Brine flushing logic
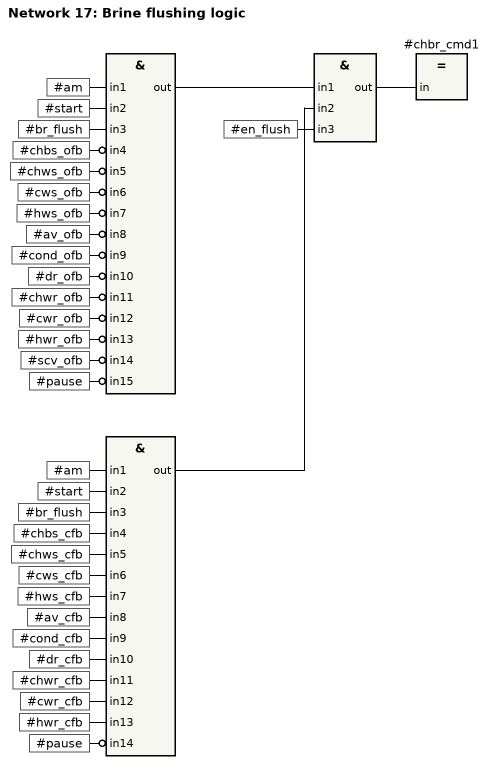
   #chbr_cmd1 := #am AND #start AND #br_flush AND NOT #chbs_ofb AND NOT #chws_ofb AND NOT #cws_ofb AND NOT #hws_ofb AND NOT #av_ofb AND NOT #cond_ofb AND NOT #dr_ofb AND NOT #chwr_ofb AND NOT #cwr_ofb AND NOT #hwr_ofb AND NOT #scv_ofb AND NOT #pause AND #am AND #start AND #br_flush AND #chbs_cfb AND #chws_cfb AND #cws_cfb AND #hws_cfb AND #av_cfb AND #cond_cfb AND #dr_cfb AND #chwr_cfb AND #cwr_cfb AND #hwr_cfb AND NOT #pause AND #en_flush;
END_REGION

REGION Network 18: Steam flushing logic
   // Steam flushing logic
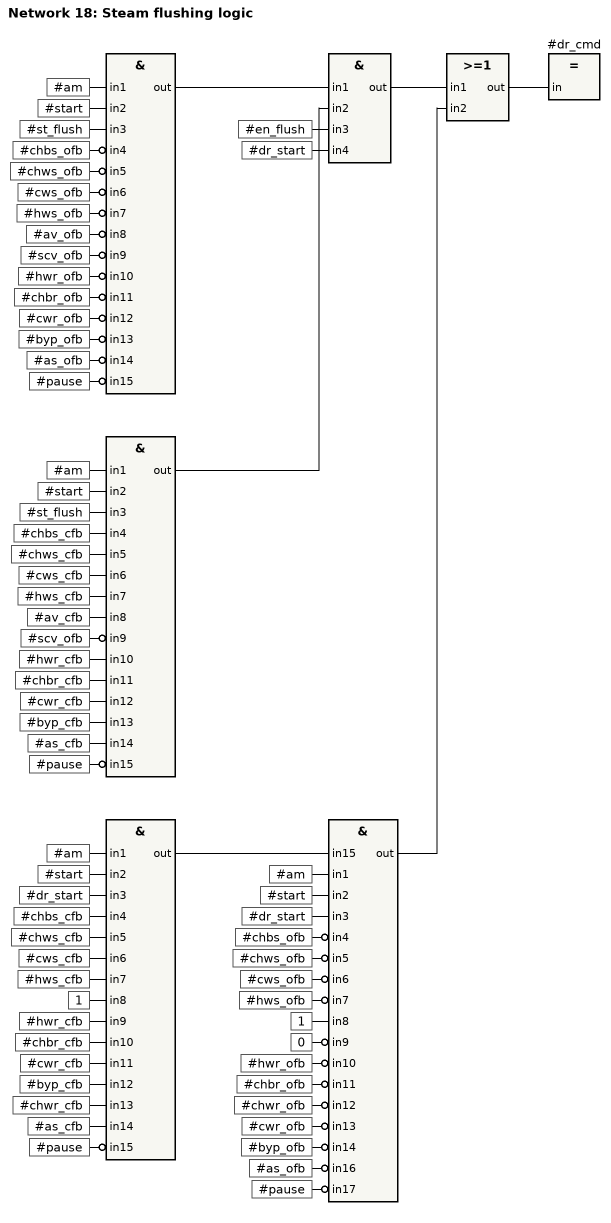
   #dr_cmd := (#am AND #start AND #st_flush AND NOT #chbs_ofb AND NOT #chws_ofb AND NOT #cws_ofb AND NOT #hws_ofb AND NOT #av_ofb AND NOT #scv_ofb AND NOT #hwr_ofb AND NOT #chbr_ofb AND NOT #cwr_ofb AND NOT #byp_ofb AND NOT #as_ofb AND NOT #pause AND #am AND #start AND #st_flush AND #chbs_cfb AND #chws_cfb AND #cws_cfb AND #hws_cfb AND #av_cfb AND NOT #scv_ofb AND #hwr_cfb AND #chbr_cfb AND #cwr_cfb AND #byp_cfb AND #as_cfb AND NOT #pause AND #en_flush AND #dr_start) OR (#am AND #start AND #dr_start AND #chbs_cfb AND #chws_cfb AND #cws_cfb AND #hws_cfb AND 1 AND #hwr_cfb AND #chbr_cfb AND #cwr_cfb AND #byp_cfb AND #chwr_cfb AND #as_cfb AND NOT #pause AND #am AND #start AND #dr_start AND NOT #chbs_ofb AND NOT #chws_ofb AND NOT #cws_ofb AND NOT #hws_ofb AND 1 AND NOT 0 AND NOT #hwr_ofb AND NOT #chbr_ofb AND NOT #chwr_ofb AND NOT #cwr_ofb AND NOT #byp_ofb AND NOT #as_ofb AND NOT #pause);
END_REGION

REGION Network 19: chw flushing logic
   // chw flushing logic
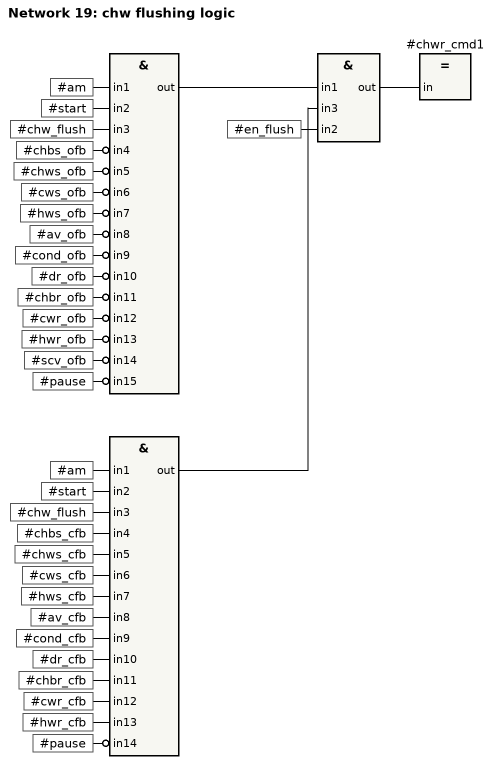
   #chwr_cmd1 := #am AND #start AND #chw_flush AND NOT #chbs_ofb AND NOT #chws_ofb AND NOT #cws_ofb AND NOT #hws_ofb AND NOT #av_ofb AND NOT #cond_ofb AND NOT #dr_ofb AND NOT #chbr_ofb AND NOT #cwr_ofb AND NOT #hwr_ofb AND NOT #scv_ofb AND NOT #pause AND #am AND #start AND #chw_flush AND #chbs_cfb AND #chws_cfb AND #cws_cfb AND #hws_cfb AND #av_cfb AND #cond_cfb AND #dr_cfb AND #chbr_cfb AND #cwr_cfb AND #hwr_cfb AND NOT #pause AND #en_flush;
END_REGION

REGION Network 20: air supply and bypass open logic
   // air supply and bypass open logic
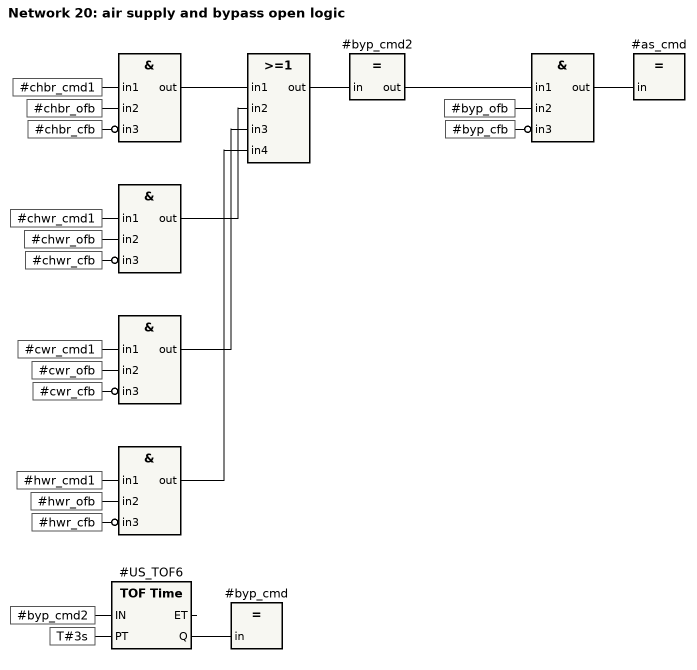
   #byp_cmd2 := (#chbr_cmd1 AND #chbr_ofb AND NOT #chbr_cfb) OR (#chwr_cmd1 AND #chwr_ofb AND NOT #chwr_cfb) OR (#cwr_cmd1 AND #cwr_ofb AND NOT #cwr_cfb) OR (#hwr_cmd1 AND #hwr_ofb AND NOT #hwr_cfb);
   #as_cmd := #byp_cmd2 AND #byp_ofb AND NOT #byp_cfb;
   #US_TOF6(IN := #byp_cmd2, PT := T#3s);   // TOF
   #byp_cmd := #US_TOF6.Q;
END_REGION

REGION Network 21: CW flushing logic
   // CW flushing logic
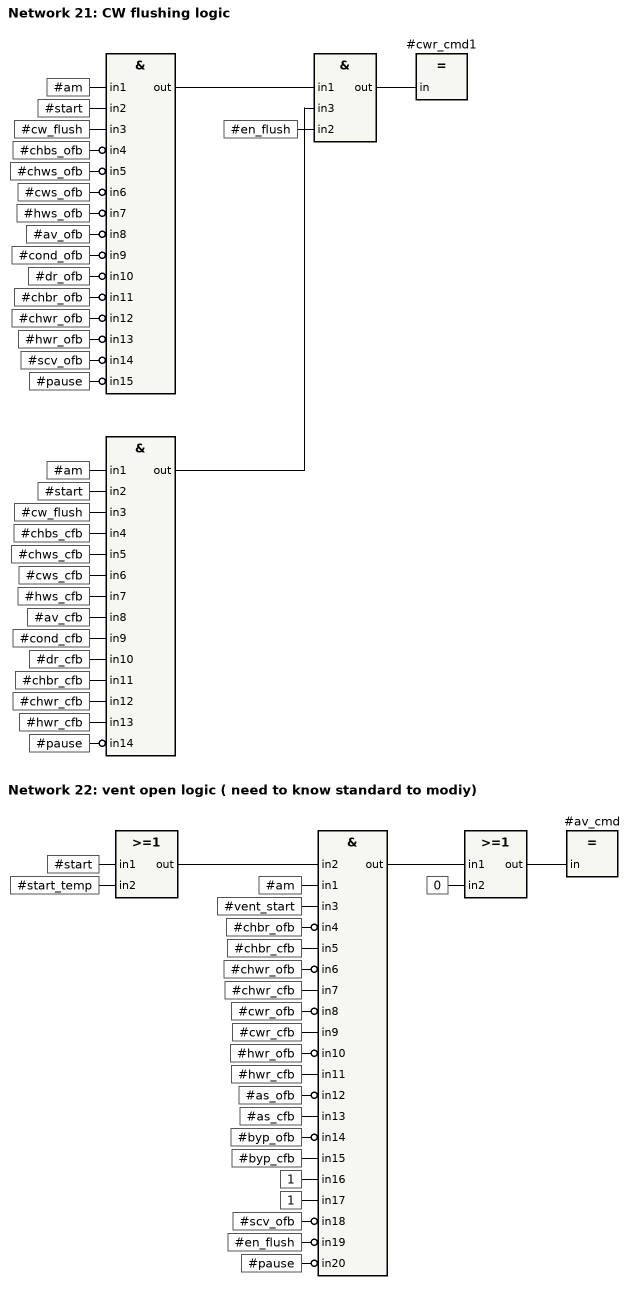
   #cwr_cmd1 := #am AND #start AND #cw_flush AND NOT #chbs_ofb AND NOT #chws_ofb AND NOT #cws_ofb AND NOT #hws_ofb AND NOT #av_ofb AND NOT #cond_ofb AND NOT #dr_ofb AND NOT #chbr_ofb AND NOT #chwr_ofb AND NOT #hwr_ofb AND NOT #scv_ofb AND NOT #pause AND #am AND #start AND #cw_flush AND #chbs_cfb AND #chws_cfb AND #cws_cfb AND #hws_cfb AND #av_cfb AND #cond_cfb AND #dr_cfb AND #chbr_cfb AND #chwr_cfb AND #hwr_cfb AND NOT #pause AND #en_flush;
END_REGION

REGION Network 22: vent open logic ( need to know standard to modiy)
   // vent open logic
   #av_cmd := ((#start OR #start_temp) AND #am AND #vent_start AND NOT #chbr_ofb AND #chbr_cfb AND NOT #chwr_ofb AND #chwr_cfb AND NOT #cwr_ofb AND #cwr_cfb AND NOT #hwr_ofb AND #hwr_cfb AND NOT #as_ofb AND #as_cfb AND NOT #byp_ofb AND #byp_cfb AND 1 AND 1 AND NOT #scv_ofb AND NOT #en_flush AND NOT #pause) OR 0;
END_REGION

REGION Network 23: hw flushing logic
   // hw flushing logic
